PROGRAM JIG002_MANSCANIA2016
VAR
END_VAR

END_PROGRAM

(* stored: Version 1.1.0.1, ProductVersion 3.1.4022.18
   POU JIG002_MANSCANIA2016: Id {ff368a16-e9de-463e-b220-2133544492e6}, SpecialFunc None *)
